{attribute 'qualified_only'}
{attribute 'strict'}
TYPE eDriveModeOfOperation :
(
	ProfilePositionMode				:= 1,
	VelocityCtrMode    				:= 2,
	ProfileVelocityMode 	   	    := 3,
	TorqueVelocityMode 				:= 4,
	HomingMode				    	:= 6,
	InterpolationPosMode			:= 7,
	CyclicSyncMode					:= 8,
	CyclicSyncVelocity				:= 9,
	CyclicSyncTorque				:= 10
	
	
);
END_TYPE

(* stored: Version 1.1.0.1, ProductVersion 3.1.4024.3
   DUT eDriveModeOfOperation: Id {357fc553-50d4-4739-9d95-cfa392d1d853} *)
